// TIA Portal project "Mała" (V17)

(* hardware
DEVICE "S7-1200 station_1"  S7-1200 Station
   slot 0: "Rack_0"  S7-1200 Rack  Rack  V1.0
   slot 1: "PLC_1"  CPU 1214C DC/DC/DC  6ES7 214-1AG40-0XB0  V4.5
*)

// ===== PLC "PLC_1"  CPU 1214C DC/DC/DC =====

VAR_GLOBAL   // PLC tag table "Default tag table"
   "System_Byte" AT %MB1 : Byte;
   "FirstScan" AT %M1.0 : Bool;
   "DiagStatusUpdate" AT %M1.1 : Bool;
   "AlwaysTRUE" AT %M1.2 : Bool;
   "AlwaysFALSE" AT %M1.3 : Bool;
   "Clock_Byte" AT %MB0 : Byte;
   "Clock_10Hz" AT %M0.0 : Bool;
   "Clock_5Hz" AT %M0.1 : Bool;
   "Clock_2.5Hz" AT %M0.2 : Bool;
   "Clock_2Hz" AT %M0.3 : Bool;
   "Clock_1.25Hz" AT %M0.4 : Bool;
   "Clock_1Hz" AT %M0.5 : Bool;
   "Clock_0.625Hz" AT %M0.6 : Bool;
   "Clock_0.5Hz" AT %M0.7 : Bool;
   "Załączenie Zespołu Hydraulicznego I" AT %I0.0 : Bool;
   "Wyłączenie Zespołu Hydraulicznego" AT %I0.1 : Bool;
   "Sterowanie 2-Ręczne" AT %I0.2 : Bool;
   "Uszkodzenie Termiczne Zespołu Hydraulicznego" AT %I0.3 : Bool;
   "Spoczynkowa Pozycja Noża" AT %I0.4 : Bool;
   "Krańcowa Pozycja Noża" AT %I0.5 : Bool;
   "Położenie Spoczynkowe Siłownika Tasaka" AT %I0.6 : Bool;
   "Zatrzymanie Awaryjne/Otwarcie Pokrywy" AT %I0.7 : Bool;
   "Głowa w Maszynie" AT %I1.0 : Bool;
   "Zabezpiecznie Głowa Nie Za Duża" AT %I1.1 : Bool;
   "Załączenie Zespołu Hydraulicznego Q" AT %Q0.0 : Bool;
   "Główny Zawór Powietrza" AT %Q0.1 : Bool;
   "Siłownik Popychacza" AT %Q0.2 : Bool;
   "Siłownik Przemieszczenia Piły" AT %Q0.3 : Bool;
   "Siłownik Odcisku Noży" AT %Q0.4 : Bool;
   "Siłownik Tasaka" AT %Q0.5 : Bool;
   "Ogólna Awaria" AT %Q0.6 : Bool;
   "MI_Załączenie Zespołu Hydraulicznego I" AT %M200.0 : Bool;
   "MI_Głowa w Maszynie" AT %M200.1 : Bool;
   "MI_Sterowanie 2-Ręczne" AT %M200.2 : Bool;
   "MQ_Załączenie Zespołu Hydraulicznego" AT %M200.3 : Bool;
   "MQ_Siłownik Popychacza" AT %M200.4 : Bool;
   "MQ_Siłownik Przemieszczenia Piły" AT %M200.5 : Bool;
   "MQ_Siłownik Odcisku Noży" AT %M200.6 : Bool;
   "MQ_Siłownik Tasaka" AT %M200.7 : Bool;
   "M_SIM" AT %M210.0 : Bool;
   "MI_Zatrzymanie Awaryjne/Otwarcie Pokrywy" AT %M201.0 : Bool;
   "MI_Wyłączenie Zespołu Hydraulicznego" AT %M201.1 : Bool;
   "MI_Uszkodzenie Termiczne Zespołu Hydraulicznego" AT %M201.2 : Bool;
END_VAR

TYPE "DT_TIME"
   STRUCT
      hours : UDInt;
      minutes : UDInt;
      seconds : UDInt;
      miliseconds : UDInt;
      nanoseconds : UDInt;
   END_STRUCT;
END_TYPE

TYPE "TonTof"
// ========== SSI Schäfer, (c)Copyright (2018) All Rights Reserved ==========
//  @Author: Johannes Hirtler 
//  @Release version: [generated release version number]
//  ==========================================================================
//  @Functionality
//  TonTof state structure provides all TonTof relevant variables
   STRUCT
      ton_tof : Bool;   // Delayed on and off
      ton : Bool;   // Delayed on
      tof : Bool;   // Delayed off
      ton_tof_re : Bool;   // Delayed on rising edge
      ton_tof_fe : Bool;   // Delayed off falling edge
      act_ton_time : "DT_TIME";   // Current time on-delay
      act_tof_time : "DT_TIME";   // Current time off-delay
   END_STRUCT;
END_TYPE

DATA_BLOCK "Zespół Cięcia Wstępnego_DB"   // DB1
{ S7_Optimized_Access := 'TRUE' }
VERSION : 0.1
// stored: InstanceOfName Zespół Cięcia Wstępnego
"Zespół Cięcia Wstępnego"
BEGIN
END_DATA_BLOCK

DATA_BLOCK "SimBlok_DB"   // DB2
{ S7_Optimized_Access := 'TRUE' }
VERSION : 0.1
// stored: InstanceOfName SimBlok
"SimBlok"
BEGIN
END_DATA_BLOCK

DATA_BLOCK "cycle_time_DB"   // DB3
{ S7_Optimized_Access := 'TRUE' }
VERSION : 0.1
// stored: InstanceOfName cycle_time
"cycle_time"
BEGIN
END_DATA_BLOCK

FUNCTION_BLOCK "Zespół Cięcia Wstępnego"   // FB1, SCL
{ S7_Optimized_Access := 'TRUE' }
VERSION : 0.1
   VAR_INPUT
      "Załączenie Zespołu Hydraulicznego I" : Bool;
      "Wyłączenie Zespołu Hydraulicznego" : Bool;
      "Sterowanie 2-Ręczne" : Bool;
      "Uszkodzenie Termiczne Zespołu Hydraulicznego" : Bool;
      "Spoczynkowa Pozycja Noża" : Bool;
      "Krańcowa Pozycja Noża" : Bool;
      "Położenie Spoczynkowe Siłownika Tasaka" : Bool;
      "Zatrzymanie Awaryjne/Otwarcie Pokrywy" : Bool;
      "Głowa w Maszynie" : Bool;
      "Zabezpiecznie Głowa Nie Za Duża" : Bool;
      "Brak Głowy / Za duża Głowa, Czas do Błędu" : Time := T#3s;
      "Opóźnienie Obrotu Noży" : Time := T#200ms;
      "Czas Docisku Tasaka" : Time := T#1s;
   END_VAR
   VAR_OUTPUT
      "Załączenie Zespołu Hydraulicznego Q" : Bool;
      "Główny Zawór Powietrza" : Bool;
      "Siłownik Popychacza" : Bool;
      "Siłownik Przemieszczenia Piły" : Bool;
      "Siłownik Odcisku Noży" : Bool;
      "Siłownik Tasaka" : Bool;
      "Ogólna Awaria" : Bool;
   END_VAR
   VAR
      Krok : Array[0..5] of Bool;
      "Numer Kroku" : Int;
      "old załączenie zespołu hydralicznego" : Bool;
      "zespół hydrauliczny" : Bool;
      "old sterowanie 2-ręczne" : Bool;
      "błąd głowy" : Bool;
      "błąd time" : TON_TIME;
      "obrót noży" : TON_TIME;
      "start obrotu noży" : TON_TIME;
      "docisk tasaka" : TON_TIME;
   END_VAR
   VAR_TEMP
      "t_załączenie zespołu hydraulicznego zbocze narastające" : Bool;
      "t_wyłączenie zespołu hydraulicznego" : Bool;
      "t_układ bezpieczny" : Bool;
      "t_sterowanie 2-ręczne zbocze narastające" : Bool;
      "t_start obrotu noży" : Bool;
      "t_koniec docisku tasaka" : Bool;
   END_VAR
   // Krok[0] := TRUE;
BEGIN
   REGION TRANZYCJE SPECJALNE
       REGION TS1 Załączenie Zespołu Hydraulicznego
           #"t_załączenie zespołu hydraulicznego zbocze narastające" :=
           #"Załączenie Zespołu Hydraulicznego I" AND
           NOT #"old załączenie zespołu hydralicznego";

           #"old załączenie zespołu hydralicznego" :=
           #"Załączenie Zespołu Hydraulicznego I";
       END_REGION

       REGION TS2 Wyłączenie Zespołu Hydraulicznego
           #"t_wyłączenie zespołu hydraulicznego" :=
           NOT #"Zatrzymanie Awaryjne/Otwarcie Pokrywy" OR
           #"Wyłączenie Zespołu Hydraulicznego" OR
           #"Uszkodzenie Termiczne Zespołu Hydraulicznego";

       END_REGION

       REGION TS3 Układ Bezpieczny
           #"t_układ bezpieczny" :=
           #"Zatrzymanie Awaryjne/Otwarcie Pokrywy" AND
           #"zespół hydrauliczny" AND
           NOT #"Uszkodzenie Termiczne Zespołu Hydraulicznego";

           //wyzwolony układ bezpieczeństwa, przerwij cykl
           IF NOT #"t_układ bezpieczny" THEN
               #"Numer Kroku" := 0;
           END_IF;
       END_REGION

       REGION T4 Sterowanie 2-ręczne Zbocze narastające 
           #"t_sterowanie 2-ręczne zbocze narastające" :=
           #"Sterowanie 2-Ręczne" AND
           NOT #"old sterowanie 2-ręczne";

           #"old sterowanie 2-ręczne" := #"Sterowanie 2-Ręczne";

       END_REGION

       REGION T5 Czas DO Błędu Za Dużej lub Braku Głowy           
           #"błąd time"(IN := #"Numer Kroku" = 2 AND
                        #"Głowa w Maszynie",
                        PT := #"Brak Głowy / Za duża Głowa, Czas do Błędu",
                        Q => #"błąd głowy");


       END_REGION
       REGION T6 Czas DO uruchomienia obrotu noży
           // Statement section REGION
           #"obrót noży"(IN := #"Numer Kroku" = 3 AND
                         NOT "Spoczynkowa Pozycja Noża" AND
                         #"Położenie Spoczynkowe Siłownika Tasaka",
                         PT := #"Opóźnienie Obrotu Noży",
                         Q => #"t_start obrotu noży");
       END_REGION

       REGION T7 
           // Statement section REGION
           #"docisk tasaka"(IN:=#"Numer Kroku" = 6 AND
                            NOT #"Położenie Spoczynkowe Siłownika Tasaka",
                            PT:=#"Czas Docisku Tasaka",
                            Q=>#"t_koniec docisku tasaka");
       END_REGION

   END_REGION



   REGION GŁÓWNA SEKWENCJA
       CASE #"Numer Kroku" OF
           0: //Układ zabezpieczony
               //układ bezpieczeństwa nie jest wzbudzony,
               //nóż i tasak są w spoczynkowej pozycji
               IF #"t_układ bezpieczny" AND
                   #"Spoczynkowa Pozycja Noża" AND
                   NOT #"Krańcowa Pozycja Noża" AND
                   #"Położenie Spoczynkowe Siłownika Tasaka" THEN
                   #"Numer Kroku" := 1;
               END_IF;
           1: //Stan gotowości do wystartowania

               //Nóż i Tasak w wyjściowej pozycji,
               //Klapa zamknięta i wciśnięty przycisk kolanowy,
               //oraz nie jest zadziałany czujnik popychacza
               IF #"Spoczynkowa Pozycja Noża" AND
                   NOT #"Krańcowa Pozycja Noża" AND
                   #"Położenie Spoczynkowe Siłownika Tasaka" AND
                   #"t_sterowanie 2-ręczne zbocze narastające" AND
                   NOT #"Zabezpiecznie Głowa Nie Za Duża" THEN
                   #"Numer Kroku" := 2;
               END_IF;

           2:  // Wyzwolony popychacz dociska głowę

               //Upłynął czas oczekiwnia na poprawną głowę, przerwij cykl
               IF #"błąd głowy" THEN
                   #"Numer Kroku" := 0;
               END_IF;

               //Czujnik popychacza i wykrycia głowy wyzwolone,
               //gdy nóż i tasak w pozycji startowej
               IF #"Zabezpiecznie Głowa Nie Za Duża" AND
                   #"Głowa w Maszynie" AND
                   #"Spoczynkowa Pozycja Noża" AND
                   NOT #"Krańcowa Pozycja Noża" AND
                   #"Położenie Spoczynkowe Siłownika Tasaka" THEN
                   #"Numer Kroku" := 3;
               END_IF;
           3:  // Przemieszczanie noży

               //opóźniony obrót noży
               IF #"t_start obrotu noży" THEN
                   #"Numer Kroku" := 4;
               END_IF;
               ;
           4:  // Obrót noży + Przemieszczenie noży

               IF NOT "Spoczynkowa Pozycja Noża" AND
                   #"Krańcowa Pozycja Noża" THEN
                   #"Numer Kroku" := 5;
               END_IF;
               ;
           5:  // Powrót Noży
               IF #"Spoczynkowa Pozycja Noża" AND
                   NOT #"Krańcowa Pozycja Noża" THEN
                   #"Numer Kroku" := 6;
               END_IF;
           6: //Docisk Tasaka

               //Przydłużony czas zadziałania Tasaka
               IF #"t_koniec docisku tasaka" THEN
                   #"Numer Kroku" := 7;
               END_IF;
           7: //Powrót Tasaka

               IF #"Położenie Spoczynkowe Siłownika Tasaka" THEN
                   #"Numer Kroku" := 0;
               END_IF;

       END_CASE;
   END_REGION

   REGION WYJŚCIA
       REGION Załączenie Zespołu Hydraulicznego
           IF #"t_wyłączenie zespołu hydraulicznego" THEN
               #"zespół hydrauliczny" := FALSE;
           ELSIF #"t_załączenie zespołu hydraulicznego zbocze narastające" THEN
               #"zespół hydrauliczny" := TRUE;
           END_IF;

           #"Załączenie Zespołu Hydraulicznego Q" :=
           #"zespół hydrauliczny";
       END_REGION

       REGION Główny Zawór Powietrza
           #"Główny Zawór Powietrza" :=
           True;
       END_REGION

       REGION Siłownik Popychacza
           #"Siłownik Popychacza" :=
           #"Numer Kroku" = 2 OR
           #"Numer Kroku" = 3 OR
           #"Numer Kroku" = 4 OR
           #"Numer Kroku" = 5 OR
           #"Numer Kroku" = 6 OR
           #"Numer Kroku" = 7;
       END_REGION

       REGION Siłownik Przemieszczenia Piły
           #"Siłownik Przemieszczenia Piły" :=
           #"Numer Kroku" = 3 OR
           #"Numer Kroku" = 4;
       END_REGION

       REGION Siłownik Odcisku Noży
           #"Siłownik Odcisku Noży" :=
           #"Numer Kroku" = 4;
       END_REGION

       REGION Siłownik Tasaka
           #"Siłownik Tasaka" :=
           #"Numer Kroku" = 6;
       END_REGION

       REGION Ogólna Awaria
           #"Ogólna Awaria" :=
           #"Uszkodzenie Termiczne Zespołu Hydraulicznego" OR
           NOT #"Zatrzymanie Awaryjne/Otwarcie Pokrywy";
       END_REGION
   END_REGION
END_FUNCTION_BLOCK

FUNCTION_BLOCK "SimBlok"   // FB2, SCL
{ S7_Optimized_Access := 'TRUE' }
VERSION : 0.1
   VAR_INPUT
      "Załączenie Zespołu Hydraulicznego" : Bool;
      "Siłownik Popychacza" : Bool;
      "Siłownik Przemieszczenia Piły" : Bool;
      "Siłownik Odcisku Noży" : Bool;
      "Siłownik Tasaka" : Bool;
   END_VAR
   VAR_OUTPUT
      "Spoczynkowa Pozycja Noża" : Bool;
      "Krańcowa Pozycja Noża" : Bool;
      "Położenie Spoczynkowe Siłownika Tasaka" : Bool;
      "Zabezpiecznie Głowa Nie Za Duża" : Bool;
   END_VAR
   VAR
      nóż_spoczynkowa_pozycja : "TonTof_timer";
      nóż_krańcowa_pozycja : "TonTof_timer";
      tasak : "TonTof_timer";
      popychacz : "TonTof_timer";
   END_VAR
BEGIN


   #nóż_spoczynkowa_pozycja(I_IN := NOT #"Siłownik Przemieszczenia Piły",
                            I_TON_SECONDS := 1);
   #"Spoczynkowa Pozycja Noża" := #nóż_spoczynkowa_pozycja.state.ton_tof;

   #nóż_krańcowa_pozycja(I_IN:= #"Siłownik Przemieszczenia Piły" AND #"Załączenie Zespołu Hydraulicznego",
                         I_TON_SECONDS:=1);

   #"Krańcowa Pozycja Noża" := #nóż_krańcowa_pozycja.state.ton_tof;

   #popychacz(I_IN:=#"Siłownik Popychacza" AND #"Załączenie Zespołu Hydraulicznego",
              I_TON_MILISECONDS:=500);
   #"Zabezpiecznie Głowa Nie Za Duża":=#popychacz.state.ton_tof;



   #tasak(I_IN:=NOT #"Siłownik Tasaka",
          I_TON_MILISECONDS:=5000,
          I_TOF_MILISECONDS:=500);
   #"Położenie Spoczynkowe Siłownika Tasaka":= #tasak.state.ton_tof;
END_FUNCTION_BLOCK

FUNCTION_BLOCK "TonTof_timer"   // FB15, SCL
{ S7_Optimized_Access := 'TRUE' }
VERSION : 0.1
   VAR_INPUT
      I_IN : Bool;   // Input for tontof
      I_RELEASE : Bool := TRUE;   // Release tontof times
      I_TON_HOURS : UDInt := 0;   // Time for on-delay
      I_TON_MINUTES : UDInt := 0;   // Time for off-delay
      I_TON_SECONDS : UDInt := 0;   // Time for off-delay
      I_TON_MILISECONDS : UDInt := 0;   // Time for off-delay
      I_TOF_HOURS : UDInt := 0;   // Time for on-delay
      I_TOF_MINUTES : UDInt := 0;   // Time for off-delay
      I_TOF_SECONDS : UDInt := 0;   // Time for off-delay
      I_TOF_MILISECONDS : UDInt := 0;   // Time for off-delay
   END_VAR
   VAR RETAIN
      state : "TonTof";   // State
   END_VAR
   VAR_TEMP
      t_ton : "DT_TIME";
      t_tof : "DT_TIME";
      t_b : Bool;
   END_VAR
BEGIN
   REGION Evaluates a Boolean variable and forms delays and edges
     // ========== SSI Schäfer, (c)Copyright (2018) All Rights Reserved ==========
     // @Author: Johannes Hirtler
     // @Release version: (generated release version number)
     // ==========================================================================
     // @Functionality
     // Evaluates a boolean variable and forms delays an edges from the delays and
     // provide this signals in the state structure.
     // The current delay time can be stopped via the input I_RELEASE. 
   END_REGION


   #t_ton := "define_time"(I_HOURS := #I_TON_HOURS, I_MINUTES := #I_TON_MINUTES, I_SECONDS := #I_TON_SECONDS, I_MILISECONDS := #I_TON_MILISECONDS);
   #t_tof := "define_time"(I_HOURS := #I_TOF_HOURS, I_MINUTES := #I_TOF_MINUTES, I_SECONDS := #I_TOF_SECONDS, I_MILISECONDS := #I_TOF_MILISECONDS);


   REGION Count delay on and off time
     IF #I_IN THEN
       // Input is true

       // Reset the delay off time
         "reset_time"(#state.act_tof_time);

         IF #I_RELEASE AND "greater_time"(Time1 := #t_ton, Time2 := #state.act_ton_time) THEN
         // Increase the on delay time
             "add_time"(CycleTimeNs:="cycle_time_DB".cycle_time_ns,
                        "Time":=#state.act_ton_time);
       END_IF;
     ELSE
       // Input is false

       // Reset the delay on time    
         "reset_time"(#state.act_ton_time);

         IF #I_RELEASE AND "greater_time"(Time1 := #t_tof, Time2 := #state.act_tof_time) THEN
         // Increase the off delay time
             "add_time"(CycleTimeNs := "cycle_time_DB".cycle_time_ns,
                        "Time" := #state.act_tof_time);
       END_IF;
     END_IF;
   END_REGION

   REGION Delay On
       IF "greater_or_equal_time"(Time1 := #state.act_ton_time, Time2 := #t_ton) AND #I_IN THEN
       // Set the delayed on signal
       #state.ton := TRUE;
     ELSE
       // Reset the delayed on signal
       #state.ton := FALSE;
     END_IF;
   END_REGION

   REGION Delay Off
       IF "greater_or_equal_time"(Time1 := #state.act_tof_time, Time2 := #t_tof) AND NOT #I_IN THEN
       // Set the delayed off signal
       #state.tof := FALSE;
     ELSE
       // Reset the delayed off signal
       #state.tof := TRUE;
     END_IF;
   END_REGION

   REGION Delay on and off
     IF #state.ton THEN
       // Set the delayed on and off signal
       #state.ton_tof := TRUE;
     ELSIF NOT #state.tof THEN
       // Reset the delayed an and off signal
       #state.ton_tof := FALSE;
     END_IF;
   END_REGION
END_FUNCTION_BLOCK

ORGANIZATION_BLOCK "Main"   // OB1, LAD, ProgramCycle
TITLE = "Main Program Sweep (Cycle)"
{ S7_Optimized_Access := 'TRUE' }
VERSION : 0.1
   VAR_INPUT
      Initial_Call : Bool;   // Initial call of this OB
      Remanence : Bool;   // =True, if remanent data are available
   END_VAR
BEGIN

REGION Network 1: Czas cyklu sterownika
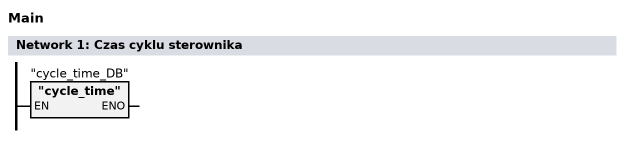
   RUNG wire#powerrail
      "cycle_time_DB"()
   END_RUNG
   // the same network as SCL:
   "cycle_time_DB"();   // "cycle_time"
END_REGION

REGION Network 2 (SCL): Symulowanie wejść
   IF "M_SIM" THEN

       "Załączenie Zespołu Hydraulicznego I" := "MI_Załączenie Zespołu Hydraulicznego I";
       "Głowa w Maszynie" := "MI_Głowa w Maszynie";
       "Sterowanie 2-Ręczne" := "MI_Sterowanie 2-Ręczne";
       "Wyłączenie Zespołu Hydraulicznego" := "MI_Wyłączenie Zespołu Hydraulicznego";
       "Zatrzymanie Awaryjne/Otwarcie Pokrywy" := "MI_Zatrzymanie Awaryjne/Otwarcie Pokrywy";
       "Uszkodzenie Termiczne Zespołu Hydraulicznego" := "MI_Uszkodzenie Termiczne Zespołu Hydraulicznego";


       "SimBlok_DB"("Załączenie Zespołu Hydraulicznego" := "MQ_Załączenie Zespołu Hydraulicznego",
                    "Siłownik Popychacza" := "MQ_Siłownik Popychacza",
                    "Siłownik Przemieszczenia Piły" := "MQ_Siłownik Przemieszczenia Piły",
                    "Siłownik Odcisku Noży" := "MQ_Siłownik Odcisku Noży",
                    "Siłownik Tasaka" := "MQ_Siłownik Tasaka",
                    "Spoczynkowa Pozycja Noża" => "Spoczynkowa Pozycja Noża",
                    "Krańcowa Pozycja Noża" => "Krańcowa Pozycja Noża",
                    "Położenie Spoczynkowe Siłownika Tasaka" => "Położenie Spoczynkowe Siłownika Tasaka",
                    "Zabezpiecznie Głowa Nie Za Duża" => "Zabezpiecznie Głowa Nie Za Duża");
   END_IF;
END_REGION

REGION Network 3 (SCL): Główny program
   "Zespół Cięcia Wstępnego_DB"("Załączenie Zespołu Hydraulicznego I":="Załączenie Zespołu Hydraulicznego I",
                                "Wyłączenie Zespołu Hydraulicznego":="Wyłączenie Zespołu Hydraulicznego",
                                "Sterowanie 2-Ręczne":="Sterowanie 2-Ręczne",
                                "Uszkodzenie Termiczne Zespołu Hydraulicznego":="Uszkodzenie Termiczne Zespołu Hydraulicznego",
                                "Spoczynkowa Pozycja Noża":="Spoczynkowa Pozycja Noża",
                                "Krańcowa Pozycja Noża":="Krańcowa Pozycja Noża",
                                "Położenie Spoczynkowe Siłownika Tasaka":="Położenie Spoczynkowe Siłownika Tasaka",
                                "Zatrzymanie Awaryjne/Otwarcie Pokrywy":="Zatrzymanie Awaryjne/Otwarcie Pokrywy",
                                "Głowa w Maszynie":="Głowa w Maszynie",
                                "Zabezpiecznie Głowa Nie Za Duża":="Zabezpiecznie Głowa Nie Za Duża",
                                "Załączenie Zespołu Hydraulicznego Q"=>"Załączenie Zespołu Hydraulicznego Q",
                                "Główny Zawór Powietrza"=>"Główny Zawór Powietrza",
                                "Siłownik Popychacza"=>"Siłownik Popychacza",
                                "Siłownik Przemieszczenia Piły"=>"Siłownik Przemieszczenia Piły",
                                "Siłownik Odcisku Noży"=>"Siłownik Odcisku Noży",
                                "Siłownik Tasaka"=>"Siłownik Tasaka",
                                "Ogólna Awaria"=>"Ogólna Awaria");
END_REGION

REGION Network 4 (SCL): Przepisanie wyjść
   IF "M_SIM" THEN
       "MQ_Załączenie Zespołu Hydraulicznego" := "Załączenie Zespołu Hydraulicznego Q";
       "MQ_Siłownik Popychacza" := "Siłownik Popychacza";
       "MQ_Siłownik Przemieszczenia Piły" := "Siłownik Przemieszczenia Piły";
       "MQ_Siłownik Odcisku Noży" := "Siłownik Odcisku Noży";
       "MQ_Siłownik Tasaka" := "Siłownik Tasaka";
   END_IF;
END_REGION
END_ORGANIZATION_BLOCK

// folder: Time

FUNCTION_BLOCK "cycle_time"   // FB4, SCL
{ S7_Optimized_Access := 'TRUE' }
VERSION : 0.1
   VAR RETAIN
      auxiliary_memory : LReal;   // Auxiliary memory
   END_VAR
   VAR
      runtime : LReal;
      cycle_time_ns : UDInt;
   END_VAR
   VAR_TEMP
      t_runtime_lreal : LReal;   // Runtime
   END_VAR
BEGIN
   #t_runtime_lreal := RUNTIME(#auxiliary_memory);
   #cycle_time_ns := #t_runtime_lreal * 1000000;
END_FUNCTION_BLOCK

FUNCTION "unit" : Void   // FC1, SCL
{ S7_Optimized_Access := 'TRUE' }
VERSION : 0.1
   VAR_INPUT
      RANGE : UDInt;
   END_VAR
   VAR_IN_OUT
      IN_UNIT : UDInt;
      OUT_UNIT : UDInt;
   END_VAR
   VAR_TEMP
      t_udint : UDInt;
   END_VAR
BEGIN
   IF #IN_UNIT >= #RANGE THEN
       #t_udint := #IN_UNIT / #RANGE;
       #IN_UNIT := #IN_UNIT MOD #RANGE;
       #OUT_UNIT := #OUT_UNIT + #t_udint;
   END_IF;
END_FUNCTION

FUNCTION "add_time" : Void   // FC2, SCL
{ S7_Optimized_Access := 'TRUE' }
VERSION : 0.1
   VAR_INPUT
      CycleTimeNs : UDInt;
   END_VAR
   VAR_IN_OUT
      "Time" : "DT_TIME";
   END_VAR
BEGIN
   #Time.nanoseconds += #CycleTimeNs;
   "unit"(RANGE := 1000,
          IN_UNIT := #Time.nanoseconds,
          OUT_UNIT := #Time.miliseconds);

   "unit"(RANGE := 1000,
          IN_UNIT := #Time.miliseconds,
          OUT_UNIT := #Time.seconds);

   "unit"(RANGE := 60,
          IN_UNIT := #Time.seconds,
          OUT_UNIT := #Time.minutes);

   "unit"(RANGE := 60,
          IN_UNIT := #Time.minutes,
          OUT_UNIT := #Time.hours);

   // "unit"(RANGE := 24,
   //        IN_UNIT := #Time.hours,
   //        OUT_UNIT := #Time.days);
END_FUNCTION

FUNCTION "reset_time" : Void   // FC3, SCL
{ S7_Optimized_Access := 'TRUE' }
VERSION : 0.1
   VAR_IN_OUT
      "Time" : "DT_TIME";
   END_VAR
BEGIN
   #Time.nanoseconds :=
   #Time.miliseconds :=
   #Time.seconds :=
   #Time.minutes :=
   #Time.hours :=
   //#Time.days :=
   0;
END_FUNCTION

FUNCTION "greater_time" : Bool   // FC4, SCL
{ S7_Optimized_Access := 'TRUE' }
VERSION : 0.1
   VAR_INPUT
      Time1 : "DT_TIME";
      Time2 : "DT_TIME";
   END_VAR
BEGIN
   IF #Time1.hours > #Time2.hours THEN
       #greater_time := TRUE;
       RETURN;
   ELSIF #Time1.hours = #Time2.hours THEN
       IF #Time1.minutes > #Time2.minutes THEN
           #greater_time := TRUE;
           RETURN;
       ELSIF #Time1.minutes = #Time2.minutes THEN
           IF #Time1.seconds > #Time2.seconds THEN
               #greater_time := TRUE;
               RETURN;
           ELSIF #Time1.seconds = #Time2.seconds THEN
               IF #Time1.miliseconds > #Time2.miliseconds THEN
                   #greater_time := TRUE;
                   RETURN;
               ELSIF #Time1.miliseconds = #Time2.miliseconds THEN
                   IF #Time1.nanoseconds > #Time2.nanoseconds THEN
                       #greater_time := TRUE;
                       RETURN;
                   ELSIF #Time1.nanoseconds = #Time2.nanoseconds THEN
                       ;
                   END_IF;
               END_IF;
           END_IF;
       END_IF;
   END_IF;
   #greater_time := FALSE;
END_FUNCTION

FUNCTION "define_time" : "DT_TIME"   // FC5, SCL
{ S7_Optimized_Access := 'TRUE' }
VERSION : 0.1
   VAR_INPUT
      I_HOURS : UDInt;
      I_MINUTES : UDInt;
      I_SECONDS : UDInt;
      I_MILISECONDS : UDInt;
   END_VAR
   VAR_TEMP
      hours : UDInt;
      minutes : UDInt;
      seconds : UDInt;
      miliseconds : UDInt;
   END_VAR
BEGIN
   "reset_time"(#define_time);

   IF #I_MILISECONDS>=1000 THEN
       #define_time.seconds := #I_MILISECONDS / 1000;
       #define_time.miliseconds := #I_MILISECONDS MOD 1000;
   ELSE
       #define_time.miliseconds:=#I_MILISECONDS;
   END_IF;

   IF #I_SECONDS+#define_time.seconds  >= 60 THEN
       #define_time.minutes := #I_SECONDS / 60;
       #define_time.seconds := (#I_SECONDS+#define_time.seconds) MOD 60;
   ELSE
       #define_time.seconds := #I_SECONDS+#define_time.seconds;
   END_IF;

   IF #I_MINUTES + #define_time.minutes >= 60 THEN
       #define_time.hours := #I_MINUTES / 60;
       #define_time.minutes := (#I_MINUTES + #define_time.minutes) MOD 60;
   ELSE
       #define_time.minutes := #I_MINUTES + #define_time.minutes;
   END_IF;

   #define_time.hours := #I_HOURS+#define_time.hours;
END_FUNCTION

FUNCTION "greater_or_equal_time" : Bool   // FC6, SCL
{ S7_Optimized_Access := 'TRUE' }
VERSION : 0.1
   VAR_INPUT
      Time1 : "DT_TIME";
      Time2 : "DT_TIME";
   END_VAR
BEGIN
   IF #Time1.hours > #Time2.hours THEN
       #greater_or_equal_time := TRUE;
       RETURN;
   ELSIF #Time1.hours = #Time2.hours THEN
       IF #Time1.minutes > #Time2.minutes THEN
           #greater_or_equal_time := TRUE;
           RETURN;
       ELSIF #Time1.minutes = #Time2.minutes THEN
           IF #Time1.seconds > #Time2.seconds THEN
               #greater_or_equal_time := TRUE;
               RETURN;
           ELSIF #Time1.seconds = #Time2.seconds THEN
               IF #Time1.miliseconds > #Time2.miliseconds THEN
                   #greater_or_equal_time := TRUE;
                   RETURN;
               ELSIF #Time1.miliseconds = #Time2.miliseconds THEN
                   IF #Time1.nanoseconds > #Time2.nanoseconds THEN
                       #greater_or_equal_time := TRUE;
                       RETURN;
                   ELSIF #Time1.nanoseconds = #Time2.nanoseconds THEN
                       #greater_or_equal_time := TRUE;
                       RETURN;
                   END_IF;
               END_IF;
           END_IF;
       END_IF;
   END_IF;
   #greater_or_equal_time := FALSE;
END_FUNCTION